Fanuc TP program (LS listing): transport_pos.ls

/PROG  TRANSPORT_POS
/ATTR
OWNER		= MNEDITOR;
COMMENT		= "";
PROG_SIZE	= 237;
CREATE		= DATE 21-05-01  TIME 14:50:44;
MODIFIED	= DATE 21-05-12  TIME 09:23:46;
FILE_NAME	= ;
VERSION		= 0;
LINE_COUNT	= 5;
MEMORY_SIZE	= 597;
PROTECT		= READ_WRITE;
TCD:  STACK_SIZE	= 0,
      TASK_PRIORITY	= 50,
      TIME_SLICE	= 0,
      BUSY_LAMP_OFF	= 0,
      ABORT_REQUEST	= 0,
      PAUSE_REQUEST	= 0;
DEFAULT_GROUP	= 1,*,*,*,*;
CONTROL_CODE	= 00000000 00000000;
/APPL

AUTO_SINGULARITY_HEADER;
  ENABLE_SINGULARITY_AVOIDANCE   : TRUE;
/MN
   1:  UFRAME_NUM=0 ;
   2:  UTOOL_NUM=4 ;
   3:   ;
   4:J PR[28:TRANSPORT POS] R[23]% FINE    ;
   5:  CALL PLCHANDSHAKE    ;
/POS
/END
